// 隐含生成代码：不要编辑
FUNCTION CheckDivDInt : DINT
VAR_INPUT
	divisor:DINT;
END_VAR

// 隐含生成代码：这里只是对代码实现的建议
{noflow}
IF divisor = 0 THEN
	CheckDivDInt:=1;
ELSE
	CheckDivDInt:=divisor;
END_IF;
{flow}

END_FUNCTION

(* stored: Version 1.1.0.1, ProductVersion 3.1.4024.9
   POU CheckDivDInt: Id {33103286-b09d-4d55-8944-980307b0c732}, SpecialFunc CheckDivInt32 *)
